Fanuc TP program (LS listing): XFRMID.LS

/PROG  XFRMID
/ATTR
OWNER		= MNEDITOR;
COMMENT		= "provided FrMid";
PROG_SIZE	= 0;
CREATE		= DATE 26-01-01  TIME 00:00:00;
MODIFIED	= DATE 26-01-01  TIME 00:00:00;
FILE_NAME	= ;
VERSION		= 0;
LINE_COUNT	= 5;
MEMORY_SIZE	= 0;
PROTECT		= READ_WRITE;
TCD:  STACK_SIZE	= 0,
      TASK_PRIORITY	= 50,
      TIME_SLICE	= 0,
      BUSY_LAMP_OFF	= 0,
      ABORT_REQUEST	= 0,
      PAUSE_REQUEST	= 0;
DEFAULT_GROUP	= 1,*,*,*,*;
CONTROL_CODE	= 00000000 00000000;
/MN
   1:  PR[AR[3]]=PR[AR[1]]    ;
   2:  PR[AR[3],1]=PR[AR[1],1]+PR[AR[2],1]    ;
   3:  PR[AR[3],1]=PR[AR[3],1]/2    ;
   4:  PR[AR[3],2]=PR[AR[1],2]+PR[AR[2],2]    ;
   5:  PR[AR[3],2]=PR[AR[3],2]/2    ;
/POS
/END
